// TIA Portal V19 export
FUNCTION "FC60_Light" : Void   // FC60, LAD
{ S7_Optimized_Access := 'TRUE' }
// stored: AutoNumber false, IsIECCheckEnabled true, SetENOAutomatically false
   VAR_TEMP
      txConditionReady : Bool;
      txFaultError : Bool;
   END_VAR
BEGIN

REGION Network 1: Condition REady
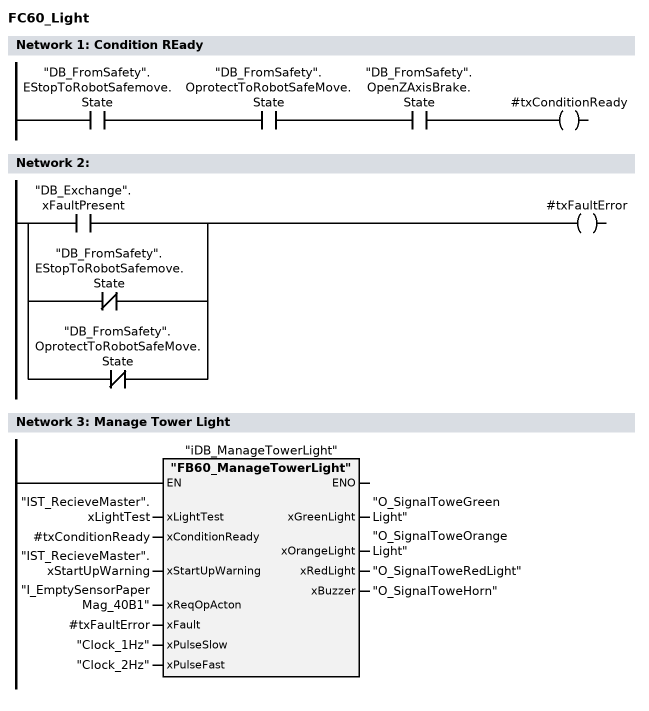
   RUNG wire#powerrail
      Contact( "DB_FromSafety".EStopToRobotSafemove.State )
      Contact( "DB_FromSafety".OprotectToRobotSafeMove.State )
      Contact( "DB_FromSafety".OpenZAxisBrake.State )
      Coil( #txConditionReady )
   END_RUNG
   // the same network as SCL:
   #txConditionReady := "DB_FromSafety".EStopToRobotSafemove.State AND "DB_FromSafety".OprotectToRobotSafeMove.State AND "DB_FromSafety".OpenZAxisBrake.State;
END_REGION

REGION Network 2
   RUNG wire#powerrail
      Contact( "DB_Exchange".xFaultPresent )
      wire#w1
      Coil( #txFaultError )
   END_RUNG
   RUNG wire#powerrail
      I_Contact( "DB_FromSafety".EStopToRobotSafemove.State )
   END_RUNG wire#w1
   RUNG wire#powerrail
      I_Contact( "DB_FromSafety".OprotectToRobotSafeMove.State )
   END_RUNG wire#w1
   // the same network as SCL:
   #txFaultError := "DB_Exchange".xFaultPresent OR NOT "DB_FromSafety".EStopToRobotSafemove.State OR NOT "DB_FromSafety".OprotectToRobotSafeMove.State;
END_REGION

REGION Network 3: Manage Tower Light
   RUNG wire#powerrail
      "iDB_ManageTowerLight"(xLightTest := "IST_RecieveMaster".xLightTest, xConditionReady := #txConditionReady, xStartUpWarning := "IST_RecieveMaster".xStartUpWarning, xReqOpActon := "I_EmptySensorPaperMag_40B1", xFault := #txFaultError, xPulseSlow := "Clock_1Hz", xPulseFast := "Clock_2Hz", xGreenLight => "O_SignalToweGreenLight", xOrangeLight => "O_SignalToweOrangeLight", xRedLight => "O_SignalToweRedLight", xBuzzer => "O_SignalToweHorn")
   END_RUNG
   // the same network as SCL:
   "iDB_ManageTowerLight"(xLightTest := "IST_RecieveMaster".xLightTest,   // "FB60_ManageTowerLight"
                          xConditionReady := #txConditionReady,
                          xStartUpWarning := "IST_RecieveMaster".xStartUpWarning,
                          xReqOpActon := "I_EmptySensorPaperMag_40B1",
                          xFault := #txFaultError,
                          xPulseSlow := "Clock_1Hz",
                          xPulseFast := "Clock_2Hz",
                          xGreenLight => "O_SignalToweGreenLight",
                          xOrangeLight => "O_SignalToweOrangeLight",
                          xRedLight => "O_SignalToweRedLight",
                          xBuzzer => "O_SignalToweHorn");
END_REGION
END_FUNCTION
